// TIA Portal V15.1 export
// export: Created 2024-06-21T08:41:07.7551582Z, ExportSetting WithDefaults, DisplayName Totally Integrated Automation Portal, DisplayVersion V15.1 Update 5, DisplayName TIA Portal Openness, DisplayVersion V15.1 Update 5, DisplayName SINAMICS Startdrive Advanced, DisplayVersion V15.1, DisplayName G130, G150, S120, S150, SINAMICS MV, S210, DisplayVersion V15.1, DisplayName G110M, G120, G120C, G120D, G120P, DisplayVersion V15.1, DisplayName STEP 7 Professional, DisplayVersion V15.1 Update 5, DisplayName STEP 7 Safety, DisplayVersion V15.1, DisplayName WinCC Professional, DisplayVersion V15.1 Update 5, DisplayName SIMATIC Visualization Architect, DisplayVersion V15.1
FUNCTION_BLOCK "LGBHooter"   // FB6659, FBD
TITLE = LRoller2W2S-MoviFitFCPN / LGBHooter
{ S7_Optimized_Access := 'TRUE' }
AUTHOR : Imtech
FAMILY : Transport
VERSION : 0.1
// =============================================================================
// This module is used in Applications when a roller one way two speed equipped 
// with SEW MOVIFIT-FC is needed. The roller can support single body tranport and 
// simultanious transport. The roller is equipped with a standard sensor setting, 
// one stop High Speed and one at the front for dual speed transport. The 
// roller uses standard handshaking signals to accomplish an infeed transfer 
// with the previous transport system and an outfeed with the next transport 
// system.
// The roller will support automatic Mode and manual Mode according specific 
// guidelines.
// The outfeed will be master over the infeed.
// Alarm "body not in Position" is also generated.
// All Alarms coming from sub-functions, TrfIn, TrfOut & LMotor2W2S-MoviFitFCPN or 
// from 
// local Alarm are summarized to give also the global Alarm A, B, C & D to 
// upper level.
// =============================================================================
// ============================================================================
// This module will start a hooter warning before the conveyor starts running or 
// when the appropriate zone goes to automode
// ============================================================================
// stored: AutoNumber false, IsIECCheckEnabled false, IsRetainMemResEnabled false, MemoryReserve 100, SetENOAutomatically False, UDAEnableTagReadback false
   VAR_INPUT
      I_AutoModeZoneWarning { ExternalAccessible := 'False'; ExternalVisible := 'False'; ExternalWritable := 'False'} : Bool;   // Mode automatic from zone warning
      I_PrevRdyToDlv { ExternalAccessible := 'False'; ExternalVisible := 'False'; ExternalWritable := 'False'} : Bool;   // Prev conveyor ready to deliver
      I_RunningReqConveyor { ExternalAccessible := 'False'; ExternalVisible := 'False'; ExternalWritable := 'False'} : Bool;   // Req cmd from conveyor
      I_StartFromRobot { ExternalAccessible := 'False'; ExternalVisible := 'False'; ExternalWritable := 'False'} : Bool;
      I_Lamptest { ExternalAccessible := 'False'; ExternalVisible := 'False'; ExternalWritable := 'False'} : Bool;   // Lamptest
      I_LampTestSteady { ExternalAccessible := 'False'; ExternalVisible := 'False'; ExternalWritable := 'False'} : Bool;   // Lamptest steady
      C_TimeHooter { ExternalAccessible := 'False'; ExternalVisible := 'False'; ExternalWritable := 'False'} : Time;   // Time of hootering
      C_TimeRunningDeadband { ExternalAccessible := 'False'; ExternalVisible := 'False'; ExternalWritable := 'False'} : Time;   // Time conveyor stops after hooring action
      C_TimeRdyToDlvInterval { ExternalAccessible := 'False'; ExternalVisible := 'False'; ExternalWritable := 'False'} : Time;   // Time interval RdyDlv
   END_VAR
   VAR_OUTPUT
      O_Hooter { ExternalAccessible := 'False'; ExternalVisible := 'False'; ExternalWritable := 'False'} : Bool;   // Hooter connection
      O_HooterReleaseConveyor { ExternalAccessible := 'False'; ExternalVisible := 'False'; ExternalWritable := 'False'} : Bool;   // Release conveyor after hootertime is finished
   END_VAR
   VAR
      TimerHooter { ExternalAccessible := 'False'; ExternalVisible := 'False'; ExternalWritable := 'False'} : TON_TIME;
      TimerDeadband { ExternalAccessible := 'False'; ExternalVisible := 'False'; ExternalWritable := 'False'} : TON_TIME;
      TimerDeadBandRdyDlv { ExternalAccessible := 'False'; ExternalVisible := 'False'; ExternalWritable := 'False'} : TON_TIME;
      HooterFinished { ExternalAccessible := 'False'; ExternalVisible := 'False'; ExternalWritable := 'False'} : Bool;
      RunningLostDelay { ExternalAccessible := 'False'; ExternalVisible := 'False'; ExternalWritable := 'False'} : Bool;
      LostRdyToDlvDelay { ExternalAccessible := 'False'; ExternalVisible := 'False'; ExternalWritable := 'False'} : Bool;
      LostRdyDlvMem { ExternalAccessible := 'False'; ExternalVisible := 'False'; ExternalWritable := 'False'} : Bool;
      LostRunningReqMem { ExternalAccessible := 'False'; ExternalVisible := 'False'; ExternalWritable := 'False'} : Bool;
      StartHooter { ExternalAccessible := 'False'; ExternalVisible := 'False'; ExternalWritable := 'False'} : Bool;
      FirstTimeRunning { ExternalAccessible := 'False'; ExternalVisible := 'False'; ExternalWritable := 'False'} : Bool;
      FirstTimeRdyDlv { ExternalAccessible := 'False'; ExternalVisible := 'False'; ExternalWritable := 'False'} : Bool;
      Edge { ExternalAccessible := 'False'; ExternalVisible := 'False'; ExternalWritable := 'False'} : Array[1..7] of Bool;   // Edge
   END_VAR
   VAR_TEMP   // added for the SCL form of the ladder/FBD networks
      _w1 : Bool;
      _w2 : Bool;
      _w3 : Bool;
      _w4 : Bool;
   END_VAR
BEGIN

REGION Network 1: **** 1 - Inputs **** HMI Commands / **** 1 - Inputs **** First program run
   // HMI Commands / First program run
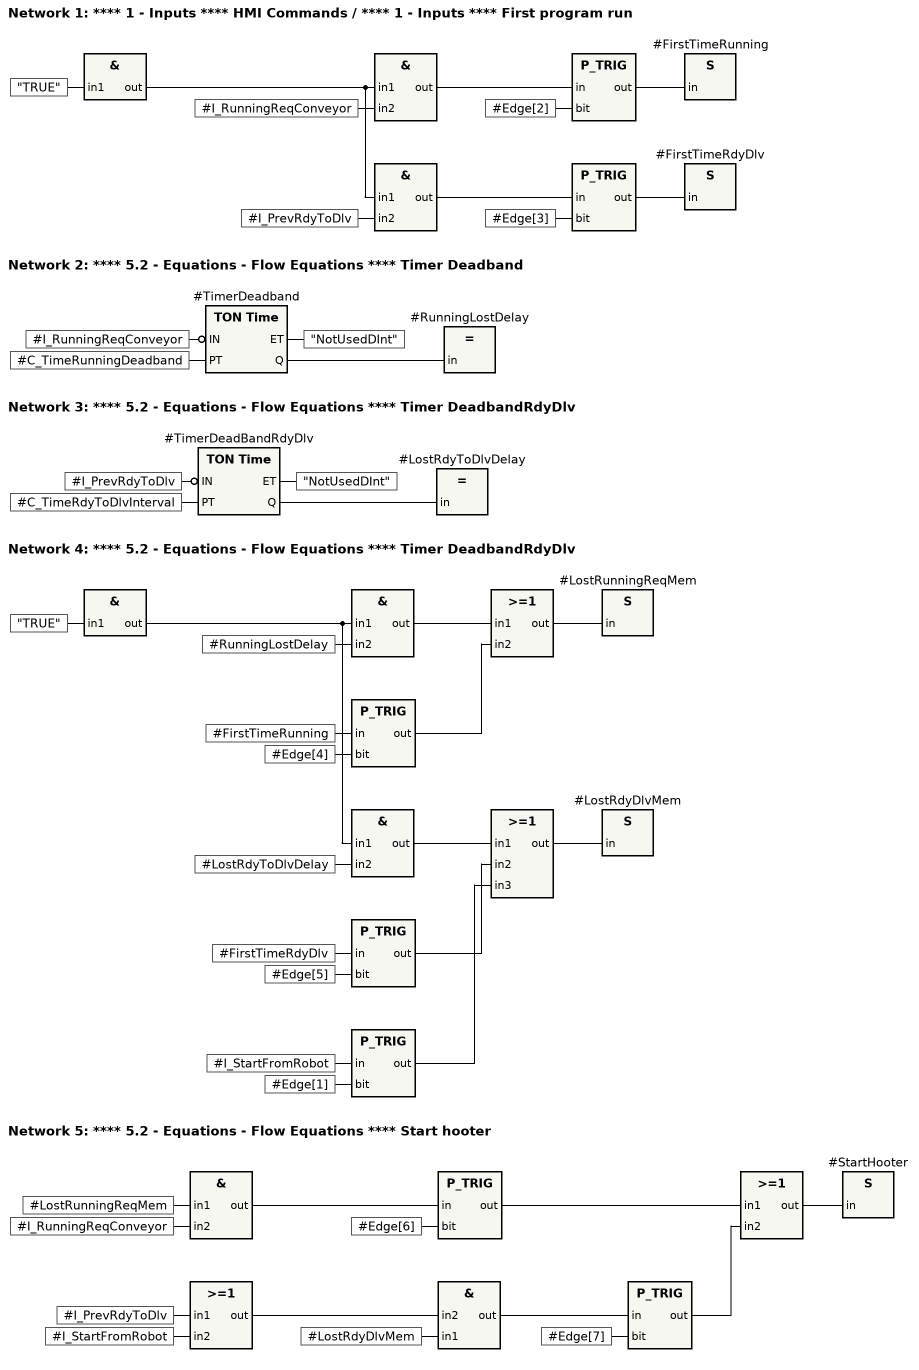
   #_w1 := "TRUE" AND #I_RunningReqConveyor;
   #_w2 := #_w1 AND NOT #Edge[2];   // rising edge
   #Edge[2] := #_w1;
   IF #_w2 THEN #FirstTimeRunning := TRUE; END_IF;
   #_w3 := "TRUE" AND #I_PrevRdyToDlv;
   #_w4 := #_w3 AND NOT #Edge[3];   // rising edge
   #Edge[3] := #_w3;
   IF #_w4 THEN #FirstTimeRdyDlv := TRUE; END_IF;
END_REGION

REGION Network 2: **** 5.2 - Equations - Flow Equations **** Timer Deadband
   // Deadband, if conveyor stop for a short time and restarts don't start the hooter.
   // Does it exceeds this time, you get a hooter alarm.
   #TimerDeadband(IN := NOT #I_RunningReqConveyor, PT := #C_TimeRunningDeadband, ET => "NotUsedDInt");   // TON
   #RunningLostDelay := #TimerDeadband.Q;
END_REGION

REGION Network 3: **** 5.2 - Equations - Flow Equations **** Timer DeadbandRdyDlv
   // Deadband, if conveyor loses ready to deliver from prev for a too long time
   #TimerDeadBandRdyDlv(IN := NOT #I_PrevRdyToDlv, PT := #C_TimeRdyToDlvInterval, ET => "NotUsedDInt");   // TON
   #LostRdyToDlvDelay := #TimerDeadBandRdyDlv.Q;
END_REGION

REGION Network 4: **** 5.2 - Equations - Flow Equations **** Timer DeadbandRdyDlv
   // Deadband, if conveyor loses ready to deliver from prev for a too long time
   #_w1 := #FirstTimeRunning AND NOT #Edge[4];   // rising edge
   #Edge[4] := #FirstTimeRunning;
   IF ("TRUE" AND #RunningLostDelay) OR #_w1 THEN #LostRunningReqMem := TRUE; END_IF;
   #_w2 := #FirstTimeRdyDlv AND NOT #Edge[5];   // rising edge
   #Edge[5] := #FirstTimeRdyDlv;
   #_w3 := #I_StartFromRobot AND NOT #Edge[1];   // rising edge
   #Edge[1] := #I_StartFromRobot;
   IF ("TRUE" AND #LostRdyToDlvDelay) OR #_w2 OR #_w3 THEN #LostRdyDlvMem := TRUE; END_IF;
END_REGION

REGION Network 5: **** 5.2 - Equations - Flow Equations **** Start hooter
   // Starting hooter conditions
   #_w1 := #LostRunningReqMem AND #I_RunningReqConveyor;
   #_w2 := #_w1 AND NOT #Edge[6];   // rising edge
   #Edge[6] := #_w1;
   #_w3 := (#I_PrevRdyToDlv OR #I_StartFromRobot) AND #LostRdyDlvMem;
   #_w4 := #_w3 AND NOT #Edge[7];   // rising edge
   #Edge[7] := #_w3;
   IF #_w2 OR #_w4 THEN #StartHooter := TRUE; END_IF;
END_REGION

REGION Network 6: **** 5.2 - Equations - Flow Equations **** Timer hooter
   // Runcommand for conveyor
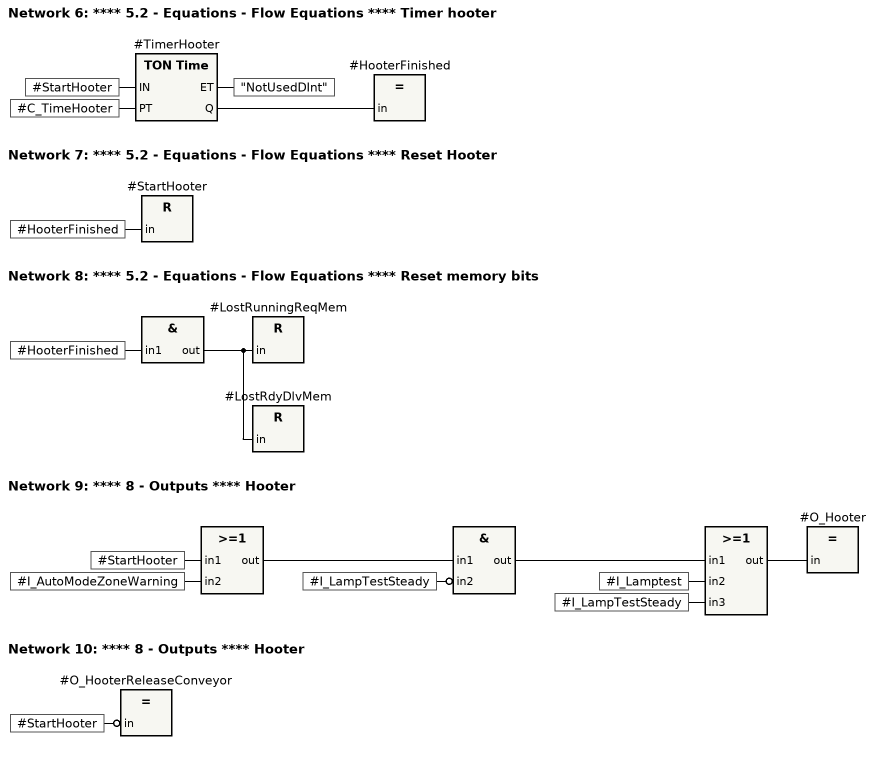
   #TimerHooter(IN := #StartHooter, PT := #C_TimeHooter, ET => "NotUsedDInt");   // TON
   #HooterFinished := #TimerHooter.Q;
END_REGION

REGION Network 7: **** 5.2 - Equations - Flow Equations **** Reset Hooter
   // To make sure the hooter goes for the SP time. Without the hooter would go with 
   // the changing of the inputsignal
   IF #HooterFinished THEN #StartHooter := FALSE; END_IF;
END_REGION

REGION Network 8: **** 5.2 - Equations - Flow Equations **** Reset memory bits
   // If hooter is finished set the memory bits
   IF #HooterFinished THEN
       #LostRunningReqMem := FALSE;
       #LostRdyDlvMem := FALSE;
   END_IF;
END_REGION

REGION Network 9: **** 8 - Outputs **** Hooter
   #O_Hooter := ((#StartHooter OR #I_AutoModeZoneWarning) AND NOT #I_LampTestSteady) OR #I_Lamptest OR #I_LampTestSteady;
END_REGION

REGION Network 10: **** 8 - Outputs **** Hooter
   #O_HooterReleaseConveyor := NOT #StartHooter;
END_REGION
END_FUNCTION_BLOCK
